Universal Robots PolyScope program: RC_E2_PLACE_230.urp

Program RC_E2_PLACE_230 (createdIn=3.0.0 lastSavedIn=3.0.0 directory=/programs installation=default)
Robot Program (runOnlyOnce=true motionType=MoveJ speed=1.047198 acceleration=1.396263 useActiveTCP=false)
  'Program generated by RoboDK v4.1.0 for UR3e_HORNO on 05/09/2022 13:30:10'
  'Using nominal kinematics.'
  'Using Ref. Frame Placas OK: p[-0.610000, 1.705000, -0.872000, 0.000000, 0.000000, 0.000000]'
  'Using TCP 0208-0001-0001-307-000-3 Horno: p[0.000000, 0.000000, 0.164750, 0.000000, 0.000000, 0.000000]'
  Script: set_tcp(p[0.000000, 0.000000, 0.164750, 0.000000, 0.000000, 0.000000])
  Script: movej([0.766615, -1.993514, -0.971187, -1.755769, 1.569310, -0.817092],0.60000,0.12500,0,0.0000)
  Script: movej([0.910270, -2.278226, -0.506229, -1.936145, 1.570482, -0.673442],0.12000,0.10000,0,0.0000)
  Script: movej([0.910270, -2.235872, -0.678644, -1.806084, 1.570482, -0.673442],0.12000,0.10000,0,0.0000)
  'Detach from 0208-0001-0001-307-000-3 Horno'
  MoveL speed 500 mm/s, acceleration 900 mm/s^2 (useActiveTCP=true)
    Waypoint Waypoint_1: TCP in base x=-235.72 y=1973 z=-718.002 mm, rx=3.1349 ry=0.0202 rz=-0.0076 rad; joints [52.155, -130.533, -29.005, -110.933, 89.982, -38.585] deg; flange x=-234.931 y=1974.1 z=-553.258 mm, rx=3.1349 ry=0.0202 rz=-0.0076 rad
  Script: movej([0.766615, -1.993514, -0.971187, -1.755769, 1.569310, -0.817092],0.90000,0.50000,0,0.0000)
